PROGRAM Axis02_Interlock
VAR
//System_Bit
	Always_ON	:	BOOL	:=TRUE	;//상시 ON 
	Always_OFF	:	BOOL	:=FALSE	;//상시 OFF
END_VAR
VAR // added by the converter: edge detectors and wires of the graphical bodies
    _w1, _w2, _w3 : BOOL;
END_VAR

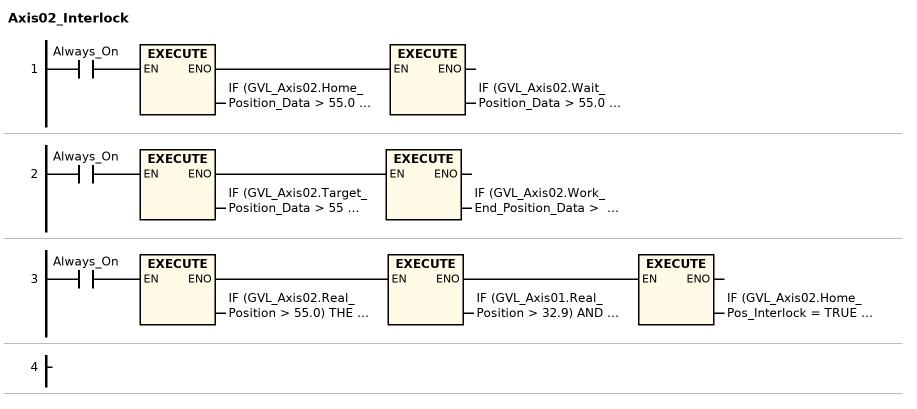
// NETWORK 1
_w1 := Always_On;
IF _w1 THEN
    IF (GVL_Axis02.Home_Position_Data > 55.0) THEN
        
        IF (GVL_Axis01.Real_Position > 1.1) AND
           (GVL_Axis04.Real_Position < 19.1) AND
           (GVL_Axis03.Real_Position >= 3.4) AND (GVL_Axis03.Real_Position <= 48) AND
           (GVL_Axis05.Real_Position >= -10.0) AND (GVL_Axis05.Real_Position <= 10.0) THEN
    
            GVL_Axis02.Home_Pos_Interlock := TRUE;
        ELSE
            GVL_Axis02.Home_Pos_Interlock := FALSE;
        END_IF;
    ELSE
        GVL_Axis02.Home_Pos_Interlock := TRUE;
    
    END_IF;
END_IF
IF _w1 THEN
    IF (GVL_Axis02.Wait_Position_Data > 55.0) THEN
        
        IF (GVL_Axis01.Real_Position > 1.1) AND
           (GVL_Axis04.Real_Position < 19.1) AND
           (GVL_Axis03.Real_Position >= 3.4) AND (GVL_Axis03.Real_Position <= 48) AND
           (GVL_Axis05.Real_Position >= -10.0) AND (GVL_Axis05.Real_Position <= 10.0) THEN
    
            GVL_Axis02.Wait_Pos_Interlock := TRUE;
        ELSE
            GVL_Axis02.Wait_Pos_Interlock := FALSE;
        END_IF;
    ELSE
        GVL_Axis02.Wait_Pos_Interlock := TRUE;
    
    END_IF;
END_IF

// NETWORK 2
_w2 := Always_On;
IF _w2 THEN
    IF (GVL_Axis02.Target_Position_Data > 55.0) THEN
        
        IF (GVL_Axis01.Real_Position > 1.1) AND
           (GVL_Axis04.Real_Position < 19.1) AND
           (GVL_Axis03.Real_Position >= 3.4) AND (GVL_Axis03.Real_Position <= 48) AND
           (GVL_Axis05.Real_Position >= -10.0) AND (GVL_Axis05.Real_Position <= 10.0) THEN
    
            GVL_Axis02.Target_Pos_Interlock := TRUE;
        ELSE
            GVL_Axis02.Target_Pos_Interlock := FALSE;
        END_IF;
    ELSE
        GVL_Axis02.Target_Pos_Interlock := TRUE;
    
    END_IF;
END_IF
IF _w2 THEN
    IF (GVL_Axis02.Work_End_Position_Data > 55.0) THEN
        
        IF (GVL_Axis01.Real_Position > 1.1) AND
           (GVL_Axis03.Real_Position >= 3.4) AND (GVL_Axis03.Real_Position <= 48) AND
            (GVL_Axis05.Real_Position >= -10.0) AND (GVL_Axis05.Real_Position <= 10.0) THEN
    
            GVL_Axis02.Work_End_Pos_Interlock := TRUE;
        ELSE
            GVL_Axis02.Work_End_Pos_Interlock := FALSE;
        END_IF;
    ELSE
        GVL_Axis02.Work_End_Pos_Interlock := TRUE;
    
    END_IF;
END_IF

// NETWORK 3
_w3 := Always_On;
IF _w3 THEN
    IF (GVL_Axis02.Real_Position > 55.0) THEN
    	GVL_Axis02.Home_ORG_Interlock	:=	TRUE ;
    ELSE
    	IF	GVL_Axis03.Home_Position OR 
    		(GVL_Axis03.Real_Position >= 3.4) AND
    		(GVL_Axis03.Real_Position <= 30.0) THEN
    	GVL_Axis02.Home_ORG_Interlock	:=	 TRUE	;
    	END_IF
    END_IF
END_IF
IF _w3 THEN
    IF (GVL_Axis01.Real_Position > 32.9) AND (GVL_Axis03.Real_Position >= -6) AND (GVL_Axis03.Real_Position <= 40)THEN
    	GVL_Calibration.Calibration_Pos_Interlock := TRUE;
    ELSE
        GVL_Calibration.Calibration_Pos_Interlock := FALSE;
    END_IF;
END_IF
IF _w3 THEN
    IF (GVL_Axis02.Home_Pos_Interlock = TRUE) AND (GVL_Axis02.Wait_Pos_Interlock = TRUE) AND (GVL_Axis02.Target_Pos_Interlock = TRUE) AND (GVL_Axis02.Work_End_Pos_Interlock = TRUE) THEN
    	GVL_Axis02.Interlock := TRUE;
    	ELSE
    	GVL_Axis02.Interlock := FALSE;	
    
    END_IF
END_IF

// NETWORK 4

END_PROGRAM

(* stored: Version 1.1.0.1, ProductVersion 3.1.4024.15
   POU Axis02_Interlock: Id {42d17d02-c8f5-405b-a8b7-936db7d763bc}, SpecialFunc None *)
